// TIA Portal V19 export
TYPE "Ax_PB"
// stored: Access Published
   STRUCT
      Bwd_Minus : Bool := FALSE;   // PB move velocity Bwd / Minus direction. If Ax handles positioning and it's homed, a moving to Min Limit is execute
      Fwd_Plus : Bool := FALSE;   // PB move velocity Fwd / Plus direction. If Ax handles positioning and it's homed, a moving to Max Limit is execute
      MoveToPos : Bool := FALSE;   // PB move to target position. Target is on HMI struct inside machine. !! Not used on FeedMachine & SpeedMachine!!
   END_STRUCT;
END_TYPE
